Fanuc KAREL source: V_DISPLAY4D.kl

PROGRAM T
%NOLOCKGROUP
VAR
 v0 : STRING[40]
 v1 : INTEGER
BEGIN
 V_DISPLAY4D(v0, v1)
END T
